# B&R Automation Studio project firstMappView
Automation Studio 4.7.5.60 SP; technology packages: mappView 5.13.1

## Configuration Config1

CPU PC_any, AutomationRuntime C4.72, Build 4.1.2, Vc V4.72.0

### Task classes (Cpu.sw)
```
Cyclic#4:
  Program <- Program.prg
```

### Hardware
```
PC : PC_any v1.1.0.0 (OrderNumber=PC)
  ConfigurationID = firstMappView_Config1
  ActivateOpcUa = 1
  OpcUaInformationModels_PV_Version = 1
SimDevice : SimDevice v1.0.0.5  [ETH1 -> PC.IF3 [Cable Type=PowerlinkCable, Length=10, Version=1.0.0.2]]
```

## Logical view

Binary libraries used (declarations not repeated): operator, runtime, astime, AsIecCon

### Package Logical/Libraries - Global libraries

- Visualisation Logical/mappView (not shown)

### Program Logical/Program (IEC)

#### Cyclic.st - Cyclic code
```iecst
PROGRAM _CYCLIC
	IF Heating THEN
		Speed := Speed + 1;
		IF Speed >= 100 THEN
			Heating := FALSE;
		END_IF
	ELSE
		Speed := Speed - 1;
		IF Speed <= 0 THEN
			Heating := TRUE;
		END_IF
	END_IF
END_PROGRAM
```

#### Init.st - Init code
```iecst
PROGRAM _INIT
	Heating := TRUE;
	Speed := 30;
	Temperature := 20.0;
END_PROGRAM
```

#### Variables.var - Local variables
```iecst
VAR
	Speed : INT;
	Temperature : REAL;
	Heating : BOOL;
END_VAR
```

Listed in the project but not available here: Logical/Global.typ, Logical/Global.var, Logical/Program/Exit.st, Logical/Program/Types.typ
